Staubli VAL3: show_progress.pgx

program show_progress(screen& x_sScreen, num x_nNum_run, num x_nNum_total, num x_nNum_row)
begin
    userPage(sScreen_ppShelf)
  title(sScreen_ppShelf,"Progree")
  gotoxy(sScreen_ppShelf,0,x_nNum_row)

  putln(sScreen_ppShelf, toString("",x_nNum_run) + "/" + toString("",x_nNum_total))
end
